// TIA Portal V19 export
TYPE "C215_STU_IF_SVLU_TYPIC"
   STRUCT
      CMD_AAN { ExternalAccessible := 'False'; ExternalVisible := 'False'; ExternalWritable := 'False'} : Bool;   // Aansturing statisch indicatiebord vluchtroute
      CMD_RES { ExternalAccessible := 'False'; ExternalVisible := 'False'; ExternalWritable := 'False'} : Bool;   // Reset van de latched storingen
   END_STRUCT;
END_TYPE
